// TIA Portal V20 export
DATA_BLOCK "TargetGlob"   // DB4
TITLE = Setta il punto di arrivo proìevisto
{ S7_Optimized_Access := 'TRUE' }
AUTHOR : Nicola
// Imposta la posizione in coordiate assolute da raggiungere
// stored: MemoryReserve 100
   VAR
      Pos : "Position";
   END_VAR
BEGIN
END_DATA_BLOCK
